# EPICS substitutions: zfhifiSup/zfhifi_field_axis.substitutions
file zfhifi_field_axis.template {

pattern {P, AXIS}
  {"\$(P)", "X"}
  {"\$(P)", "Y"}
  {"\$(P)", "Z"}
}
